{attribute 'qualified_only'}
{attribute 'strict'}
{attribute 'to_string'}
TYPE E_MachineStatusSignaallamp :
(
	Idle := 0, // Machine staat in rustpositie
	Running,  // Machine is in beweging
	Error,   // Machine is in storing
	Resetting // Machine is aan het resetten
);
END_TYPE

(* stored: Version 1.1.0.1
   DUT E_MachineStatusSignaallamp: Id {eac53a6b-b57c-48f7-9b0e-db19503b7dc8} *)
